FUNCTION_BLOCK FB_NAME IMPLEMENTS I_NAME
VAR_INPUT
END_VAR
VAR_OUTPUT
END_VAR
VAR
	m_name : STRING := 'User';
END_VAR

{warning 'add property implementation'}
PROPERTY Name : STRING
GET
Name := m_name;
END_GET
SET
m_name := Name;
END_SET
END_PROPERTY

{warning 'add method implementation '}
METHOD NUM : INT
NUM := LEN(m_name);
END_METHOD

END_FUNCTION_BLOCK

(* stored: Version 1.1.0.1, ProductVersion 3.1.4024.3
   POU FB_NAME: Id {6065e354-1a05-4951-89a0-632450cfdc72}, SpecialFunc None
   Property Name: Id {5134a08f-f1f4-4615-ba9d-b2beb341aced}
   Get Get: Id {0513b7b3-99f5-4c87-8f0f-784bb4c25382}
   Set Set: Id {12196984-e221-4b12-a66b-356157a167b0}
   Method NUM: Id {0d51eca5-f55c-4988-9e77-8cd2ef944f9d} *)
